FUNCTION_BLOCK FB_TableVacuum
VAR_INPUT
	vacuum_measured			:LREAL;//	Pa
	vacuum_min				:LREAL:=3.5;	//	Pa 3.5
	vacuum_max				:LREAL:=10;	//	Pa	10
	setpoint				:LREAL:=6;	//	Pa	6[0-8]
	vacuum_offset_collector	:LREAL;	//	Pa	Offset used to calibrate the vacuum sensor of the vacuum collector
	setpoint_range_pct		:LREAL:=70;	//	%  Threshold used to indicate the table vacuum is ready
	vacuum_timeout			:LREAL:=6000;	//ms	TIME needed TO reach the vacuum setpoint.
	vacuum_off_timeout		:LREAL:=3000;	//	ms 	Time to turn off the vacuum
	IO_Error				:BOOL;
END_VAR
VAR_OUTPUT
	state					:INT;
	error_code					:INT;
	Run						:BOOL;
	error					:BOOL;
END_VAR
VAR
	step					:INT;
	setpoint_act			:LREAL;
	reach_setpoint_ton		:ton;
	turn_off_ton			:TON;
	turn_on_delay           :Tc2_Standard.TON;
	temp_setpoint			:LREAL;
END_VAR
VAR_IN_OUT
	Initialize				:BOOL;
	SetVacuumOn				:BOOL;
	SetVacuumOff			:BOOL;
	Setoff					:BOOL;
END_VAR


CASE step OF 
0://waiting
	IF Initialize THEN 
		step:=5;
	ELSIF SetVacuumOn THEN 
		step:=10;
	ELSIF SetVacuumOff THEN 
		step:=30;
	ELSIF Setoff OR GVL.Reset THEN 
		step:=50;
	END_IF	
5://off
	Run:=FALSE;
	setpoint_act:=0;
	SetVacuumOn:=FALSE;
	SetVacuumOff:=FALSE;
	Setoff:=FALSE;
	
	
	state:=TabVacStateEnum.off;
	error_code:=TabVacErrorEnum.no_error;
	
	IF Initialize AND 
		setpoint_range_pct<>0 AND vacuum_min>=0 AND vacuum_max>0 THEN 
		Initialize:=FALSE;
		state:=TabVacStateEnum.idle;	
		step:=0;
	END_IF
	
10://INI
	SetVacuumOff:=FALSE;			
	IF setpoint>=vacuum_min AND setpoint<=vacuum_max AND vacuum_timeout>0  THEN 
		setpoint_act:=setpoint;
	ELSIF  setpoint>=vacuum_max THEN 
			setpoint_act:=vacuum_max;
	ELSIF setpoint<=vacuum_min THEN 
		setpoint_act:=vacuum_min;
	END_IF

	IF SetVacuumOn THEN 
			step:=20;
	ELSIF Setoff THEN 
			step:=50;
	END_IF

20://waiting_vacuum_on
	SetVacuumOn:=FALSE;
	Initialize:=FALSE;
	SetVacuumOff:=FALSE;
	
	state:=TabVacStateEnum.waiting_vacuum_on;
	Run:=TRUE;
	reach_setpoint_ton(IN:=TRUE , PT:=LREAL_TO_TIME(vacuum_timeout) , Q=> , ET=> );
	IF reach_setpoint_ton.Q (*AND vacuum_measured/setpoint_act*100<setpoint_range_pct *)THEN		
		error_code:=TabVacErrorEnum.vacuum_on_timeout;
		step:=100;
	END_IF
	(*************转on 用时间******************************)
	(*IF NOT reach_setpoint_ton.Q AND  vacuum_measured/setpoint_act*100>=setpoint_range_pct THEN 	
		reach_setpoint_ton(IN:=FALSE); 		
		state:=TabVacStateEnum.on;	
		step:=0;
	END_IF*)
	
	turn_on_delay(IN:=TRUE , PT:=INT_TO_TIME(HMI_Vac_dely_on), Q=> , ET=> );
	IF NOT reach_setpoint_ton.Q AND  turn_on_delay.Q THEN 	
		reach_setpoint_ton(IN:=FALSE); 	
		turn_on_delay(IN:=FALSE);	
		state:=TabVacStateEnum.on;	
		step:=0;
	END_IF
	
	IF Setoff THEN 
		step:=50;
	END_IF
	
30://on		
	IF SetVacuumOff AND vacuum_off_timeout>0 THEN 
		step:=40;
	ELSIF Setoff THEN 
		step:=50;	
	END_IF
40://waiting_vacuum_off
	Initialize:=FALSE;
	SetVacuumOn:=FALSE;
	Setoff:=FALSE;
	
	SetVacuumOff:=FALSE;
	state:=TabVacStateEnum.waiting_vacuum_off;
	Run:=FALSE;
	turn_off_ton(IN:=TRUE , PT:=LREAL_TO_TIME(vacuum_off_timeout) , Q=> , ET=> );	 
	IF vacuum_measured<setpoint*0.5 AND NOT turn_off_ton.Q  THEN 
		turn_off_ton(IN:=FALSE);
		state:=TabVacStateEnum.idle;
		step:=0;
	ELSIF vacuum_measured>=0 AND turn_off_ton.Q THEN 
		error_code:=TabVacErrorEnum.vacuum_off_timeout;
		step:=100;
	END_IF
50://waiting_off
	Initialize:=FALSE;
	SetVacuumOn:=FALSE;
	SetVacuumOff:=FALSE;

	Setoff:=FALSE;
	state:=TabVacStateEnum.waiting_off;
	error_code:=TabVacErrorEnum.no_error;
	Run:=FALSE;
	error:=FALSE;
	
	IF vacuum_measured<=0.5 THEN 
		state:=TabVacStateEnum.off;
		step:=0;
	END_IF
100://error
	Initialize:=FALSE;
	SetVacuumOn:=FALSE;
	SetVacuumOff:=FALSE;
	
	error:=TRUE;
	state:=TabVacStateEnum.error;
	Run:=FALSE;
	reach_setpoint_ton(IN:=FALSE);
	turn_off_ton(IN:=FALSE);
	step:=0;	
END_CASE

IF Setoff OR GVL.Reset THEN 
	step:=50;
END_IF	
	
IF state<>TabVacStateEnum.off AND state<>TabVacStateEnum.waiting_off AND state<>TabVacStateEnum.error THEN 
	IF IO_Error THEN 
		error_code:=TabVacErrorEnum.unknown_error;
		step:=100;
	END_IF
	IF GVL.Emstop_Button THEN 
		error_code:=TabVacErrorEnum.emergency_error;	
		step:=100;
	END_IF
END_IF

END_FUNCTION_BLOCK

(* stored: Version 1.1.0.1, ProductVersion 3.1.4024.11
   POU FB_TableVacuum: Id {86869c7f-8e8d-44f2-8aae-98562e0f5fc2}, SpecialFunc None *)
